(* IEC 61131-3 sources: ATCMcontrol_Engineering/src/COM/softing/fc/AddOns/Softing/4CPCTarget/Libs/ATCM_System, 28 files *)

(* ---- ClearLocalTaskErrno.st ---- *)
(*[[
    UserURL= "ATCM:ClearLocalTaskErrno.htm"
]]*)
(*
 *  ATCMControl Standard Function ClearLocalTaskErrno
 *  Purpose: Clears the error state of the given task.
 *)
FUNCTION ClearLocalTaskErrno
VAR_INPUT
    NAME : ANY_STRING;
END_VAR

overload (WSTRING) inline{((COM.softing.fc.CC.system.ITask)globals.getObject(%1.toLowerCase())).setErrorNumber(0)}

END_FUNCTION

(* ---- ClearTaskErrno.st ---- *)
(*[[
    UserURL= "ATCM:ClearTaskErrno.htm"
]]*)
(*
 *  ATCMControl Standard Function ClearTaskErrno
 *  Purpose: Clears the error state variable of the
 *           calling task. Error numbers <>0 signal an
 *           error.
 *)
FUNCTION ClearTaskErrno

inline{tc.setErrorNumber(0)}

END_FUNCTION

(* ---- ColdStartInstance.st ---- *)
(*
 * ATCMControl standard function ColdStartInstance
 * ----------------------------------------------------------------------------
 * PURPOSE: initialises all program, function block or structure instance members
 *          to their coldstart initial values. This includes also all nested
 *          function blocks and structs.
     *          The function returns if the initialisation is complete.
 *
 * EXAMPLE: StopLocalTask("Task1");
 *          ColdStartInstance("Prog1.myFB");
 *
 * NOTE:    It is recommended to stop the task(s) that operates on "Prog1.myFB"
 *          before calling ColdStartInstance.
 *
 * WARNING: use this function only rarely, it may take a long time to coldstart a
 *          huge and deeply nested instance, that could cause watchdog error in the
 *          calling task. Typically this function is used in a task that also
 *          starts/stops other Tasks and therefore SetSystemTask() was called to
 *          disable the watchdog anyway.
 *)
FUNCTION ColdStartInstance
VAR_INPUT
    instPath : WSTRING;
END_VAR

NATIVE
    int    i = 0;
    Object o = null;
    java.util.StringTokenizer st = new java.util.StringTokenizer(_instpath.toLowerCase(), ".");
    while (st.hasMoreTokens())
    {
        if (i == 0)
            o = ((ObjectDirectory)((FcObject)tc).getParent()).getObject(st.nextToken());
        else
            o = ((ObjectDirectory)o).getObject(st.nextToken());

        if (o == null)
            break;

        i++;
    }

    if (o == null || !(o instanceof ObjectDirectoryEx))
    {
        DebugManager.print("error E1056: ColdStartInstance: instance path '" + _instpath + "' does not exist.");
        return;
    }
    ObjectDirectoryEx od = (ObjectDirectoryEx)o;

    try{
        for(i=0; ;i++)
        {
            FcObject          fobj = od.getObjectByID(i);
            ObjectDescriptor  odescr = fobj.getOD();
            String            init = odescr.getInitString();

            if(init != null)
            {
                //DebugManager.print("vorher="+init);
                if(init.length()==0)
                {
                    init = null;//should not happen...
                }
                else if(init.charAt(0)=='%' && !(fobj instanceof COM.softing.fc.CC.system.StringVar))
                {
                    if(init.charAt(1)=='I')
                        continue;

                    int iPos = init.indexOf('|');
                    if(iPos>0 && iPos+1<init.length())
                    {
                        init = init.substring(iPos+1);
                    }
                    else
                    {
                        init = null;
                    }
                }
                //DebugManager.print("nachher="+init);
            }

            if (fobj instanceof FcBool)
            {
                ((FcBool)fobj).putBool(init==null ? false : init.equalsIgnoreCase("true"));
            }
            else if (fobj instanceof FcInt)
            {
                ((FcInt)fobj).putInt(init==null ? 0 : Integer.parseInt(init));
            }
            else if (fobj instanceof FcLong)
            {
              ((FcLong)fobj).putLong(init==null ? 0 : Long.parseLong(init));
            }
            else if (fobj instanceof FcDouble)
            {
              ((FcDouble)fobj).putDouble(init==null ? 0 : (new Double(init)).doubleValue());
            }
            else if (fobj instanceof FcString)
            {
              ((FcString)fobj).putString(init==null ? "" : init);
            }
            else if (fobj instanceof ObjectDirectoryEx)
            {
              _F_coldstartinstance(_instpath + "."+ fobj.getOD().getName(), globals, tc);
            }
            else
            {
               throw new ClassCastException("4CC : fatal error E0041: ColdStartInstance: unknown basic type class");
            }
        }
    }catch(ArrayIndexOutOfBoundsException e)
    {
        //normal end for loop: because there is no od.getLength() !!
    }
END_NATIVE;

END_FUNCTION

(* ---- DebugBreak.st ---- *)
(*[[
    UserURL= "ATCM:DebugBreak.htm"
]]*)
(*
 *  ATCMControl Standard Function DebugBreak
 *  Purpose: break into the debugger (only if one is attached)
 *)
FUNCTION DebugBreak
VAR_INPUT
    IN : BOOL; (* break only if IN = TRUE *)
END_VAR

inline{if(%1)tc.userBreak(this)}

END_FUNCTION

(* ---- EnableTaskStatistic.st ---- *)
(*[[
    UserURL= "ATCM:EnableTaskStatistic.htm"
]]*)
(*
 *  ATCMControl Standard Function EnableTaskStatistic
 *  Purpose: Enable/Disable the automatic task
 *  statistic output of all tasks.
 *  The default after a download or coldstart or
 *  warmstart is enable=true.
 *
 *  EnableTaskStatistic(true) : enable  task statistics
 *  EnableTaskStatistic(false): disable task statistics
 *)
FUNCTION EnableTaskStatistic
VAR_INPUT
    ENABLE     : BOOL;  (* enable/disable input *)
END_VAR

inline{tc.enableTaskStatistic(%1)}

END_FUNCTION

(* ---- GetComputerName.st ---- *)
(*
    Purpose: Gets the computername of the local PC.
*)
FUNCTION GetComputerName : WSTRING
NATIVE

    try{
        java.net.InetAddress  iaddr = java.net.InetAddress.getLocalHost();
        _getcomputername = iaddr.toString() ;//yields myPC1[.dhcp.softing.com]/129.26.193.3
        //if WinNT: strip .dhcp.softing.com (win2K does not need ??..)
        int idx = Math.min(_getcomputername.lastIndexOf('/'), _getcomputername.indexOf('.'));
        if(idx>0)
            _getcomputername = _getcomputername.substring(0, idx);
    }catch(java.net.UnknownHostException e)
    {
        _getcomputername = e.toString();
    }

END_NATIVE;

END_FUNCTION

(* ---- getCurrentDateAndTime.st ---- *)
(*[[
    UserURL= "ATCM:getCurrentDateAndTime.htm"
]]*)

FUNCTION getCurrentDateAndTime : DT

inline{java.lang.System.currentTimeMillis()}

END_FUNCTION

(* ---- GetLocalTaskErrno.st ---- *)
(*[[
    UserURL= "ATCM:GetLocalTaskErrno.htm"
]]*)
(*
 *  ATCMControl Standard Function GetLocalTaskErrno
 *  Purpose: get the task error number of the named task.
 *
 *  possible return values are (among others):
 *  NO_ERROR            = 0
 *  DEADLOCK_DETECTED   = 2
 *  RUNTIME_EXCEPTION   = 3
 *)
FUNCTION GetLocalTaskErrno : DINT
VAR_INPUT
    NAME : ANY_STRING;
END_VAR

overload DINT(WSTRING) inline{((COM.softing.fc.CC.system.ITask)globals.getObject(%1.toLowerCase())).itGetTaskErrNo()}

END_FUNCTION

(* ---- GetLocalTaskState.st ---- *)
(*[[
    UserURL= "ATCM:GetLocalTaskState.htm"
]]*)
(*
 *  ATCMControl Standard Function GetLocalTaskState
 *  Purpose: get the current task execution state of the named task.
 *
 *  possible return values are:
 *  STATE_ERROR       = -1
 *  STATE_ONCREATION  = 0
 *  STATE_STOPPED     = 1
 *  STATE_RUNNING     = 2
 *  STATE_BREAK       = 3
 *)
FUNCTION GetLocalTaskState : DINT
VAR_INPUT
    NAME : ANY_STRING;
END_VAR

overload DINT(WSTRING) inline{((COM.softing.fc.CC.system.ITask)globals.getObject(%1.toLowerCase())).itGetTaskState()}

END_FUNCTION

(* ---- GetTaskErrno.st ---- *)
(*[[
    UserURL= "ATCM:GetTaskErrno.htm"
]]*)
(*
 *  ATCMControl Standard Function GetTaskErrno
 *  Purpose: returns the last error number of the
 *           calling task. Error numbers <>0 signal an
 *           error.
 *)
FUNCTION GetTaskErrno : DINT

inline{tc.getErrorNumber()}

END_FUNCTION

(* ---- getTimeSinceSystemBoot.st ---- *)
(*[[
    UserURL= "ATCM:getTimeSinceSystemBoot.htm"
]]*)

FUNCTION getTimeSinceSystemBoot : TIME

inline{DebugManager.getSystemTime()}

END_FUNCTION

(* ---- OutputDebugString.st ---- *)
(*[[
    UserURL= "ATCM:OutputDebugString.htm"
]]*)
(*
 *  ATCMControl Standard Functionblock OutputDebugString
 *  Purpose: Write a string to the control's standard output
 *           and the log file. A new line character is added
 *           automatically.
 *)
FUNCTION OutputDebugString
VAR_INPUT
    STR        : ANY_STRING;     (* a one-line message to the user*)
END_VAR

overload (wstring) inline{DebugManager.print(%1 + "\n")}
(* TODO : string *)

END_FUNCTION

(* ---- ReadControlVarBOOL.st ---- *)
(*[[
]]*)
(*
 * ATCMControl standard function ReadControlVarBOOL
 * ----------------------------------------------------------------------------
 * PURPOSE: read from a named control variable.
 *
 * EXAMPLE: bValue := ReadControlVarBOOL("Prog1.myFB.aBool);
 *
 * RETURN:  if the function fails, a OutputDebugString
 *          is made and return is FALSE.
 *
 * WARNING: use this function only rarely, it is not efficient.
 *)
FUNCTION ReadControlVarBOOL : BOOL
VAR_INPUT
   sPath : WSTRING;     (* full qualified name of the variable to read *)
END_VAR

    ReadControlVarBOOL := FALSE;

    NATIVE
        int    i = 0;
        Object o = null;

        java.util.StringTokenizer st = new java.util.StringTokenizer(_spath.toLowerCase(), ".");
        while (st.hasMoreTokens())
        {
            if (i == 0)
                o = ((ObjectDirectory)((FcObject)tc).getParent()).getObject(st.nextToken());
            else
                o = ((ObjectDirectory)o).getObject(st.nextToken());

            if (o == null)
                break;

            i++;
        }

        if (o != null)
        {
            if (o instanceof FcBool)
            {
                _readcontrolvarbool = ((FcBool)o).getBool();
            }
            else
            {
                DebugManager.print("4C_Control(ReadControlVarBOOL): variable '" + _spath + "' is not a JAVA boolean.");
            }
        }
        else
        {
            DebugManager.print("4C_Control(ReadControlVarBOOL): variable '" + _spath + "' does not exist.");
        }
    END_NATIVE;
END_FUNCTION

(* $Header: /ABK4191 Liebherr Pruefstand-Modernisierung/4C-Basis/4C_Control/ReadControlVarBOOL.st 4     13.02.02 11:15 Go $
*----------------------------------------------------------------------------*
*
* =FILENAME            $Workfile: ReadControlVarBOOL.st $
*                       $Logfile: /ABK4191 Liebherr Pruefstand-Modernisierung/4C-Basis/4C_Control/ReadControlVarBOOL.st $
*
* =PROJECT             ABK4191 Liebherr Prüfstand-Modernisierung
*
* =COMPONENT           4C_Control Library
*
* =CURRENT      $Date: 13.02.02 11:15 $
*           $Revision: 4 $
*             $Author: Go $
*----------------------------------------------------------------------------*
*******************************************************************************
*)

(* ---- ReadControlVarDINT.st ---- *)
(*[[
]]*)
(*
 * ATCMControl standard function ReadControlVarDINT
 * ----------------------------------------------------------------------------
 * PURPOSE: read from a named control variable.
 *
 * EXAMPLE: aInt := ReadControlVarDINT("Prog1.myFB.aInt);
 *
 * RETURN:  if the function fails, a OutputDebugString
 *          is made and return is 0.
 *
 * WARNING: use this function only rarely, it is not efficient.
 *)
FUNCTION ReadControlVarDINT : DINT
VAR_INPUT
   sPath : WSTRING;     (* full qualified name of the variable to read *)
END_VAR

    ReadControlVarDINT := 0;

    NATIVE
        int    i = 0;
        Object o = null;

        java.util.StringTokenizer st = new java.util.StringTokenizer(_spath.toLowerCase(), ".");
        while (st.hasMoreTokens())
        {
            if (i == 0)
                o = ((ObjectDirectory)((FcObject)tc).getParent()).getObject(st.nextToken());
            else
                o = ((ObjectDirectory)o).getObject(st.nextToken());

            if (o == null)
                break;

            i++;
        }

        if (o != null)
        {
            if (o instanceof FcInt)
            {
                _readcontrolvardint = ((FcInt)o).getInt();
            }
            else
            {
                DebugManager.print("4C_Control(ReadControlVarDINT): variable '" + _spath + "' is not a JAVA int.");
            }
        }
        else
        {
            DebugManager.print("4C_Control(ReadControlVarDINT): variable '" + _spath + "' does not exist.");
        }
    END_NATIVE;
END_FUNCTION

(* ---- ReadControlVarLINT.st ---- *)
(*[[
]]*)
(*
 * ATCMControl standard function ReadControlVarLINT
 * ----------------------------------------------------------------------------
 * PURPOSE: read from a named control variable.
 *
 * EXAMPLE: aLreal := ReadControlVarLINT("Prog1.myFB.aLint");
 *
 * RETURN:  if the function fails, a corresponding
 *          OutputDebugString is made and return is 0.
 *
 * WARNING: use this function only rarely, it is not efficient.
 *)
FUNCTION ReadControlVarLINT : LINT
VAR_INPUT
   sPath : WSTRING;     (* full qualified name of the variable to read *)
END_VAR

    ReadControlVarLINT := 0;

    NATIVE
        int    i = 0;
        Object o = null;

        java.util.StringTokenizer st = new java.util.StringTokenizer(_spath.toLowerCase(), ".");
        while (st.hasMoreTokens())
        {
            if (i == 0)
                o = ((ObjectDirectory)((FcObject)tc).getParent()).getObject(st.nextToken());
            else
                o = ((ObjectDirectory)o).getObject(st.nextToken());

            if (o == null)
                break;

            i++;
        }

        if (o != null)
        {
            if (o instanceof FcLong)
            {
                _readcontrolvarlint = ((FcLong)o).getLong();
            }
            else
            {
                DebugManager.print("4C_Control(ReadControlVarLINT): variable '" + _spath + "' is not a JAVA long.");
            }
        }
        else
        {
            DebugManager.print("4C_Control(ReadControlVarLINT): variable '" + _spath + "' does not exist.");
        }
    END_NATIVE;

END_FUNCTION

(* ---- ReadControlVarLREAL.st ---- *)
(*[[
]]*)
(*
 * ATCMControl standard function ReadControlVarLREAL
 * ----------------------------------------------------------------------------
 * PURPOSE: read from a named control variable.
 *
 * EXAMPLE: aLreal := ReadControlVarLREAL("Prog1.myFB.aLreal");
 *
 * RETURN:  if the function fails, a OutputDebugString
 *          is made and return is 0.
 *
 * WARNING: use this function only rarely, it is not efficient.
 *)
FUNCTION ReadControlVarLREAL : LREAL
VAR_INPUT
   sPath : WSTRING;     (* full qualified name of the variable to read *)
END_VAR

    ReadControlVarLREAL := 0.0;

    NATIVE
        int    i = 0;
        Object o = null;

        java.util.StringTokenizer st = new java.util.StringTokenizer(_spath.toLowerCase(), ".");
        while (st.hasMoreTokens())
        {
            if (i == 0)
                o = ((ObjectDirectory)((FcObject)tc).getParent()).getObject(st.nextToken());
            else
                o = ((ObjectDirectory)o).getObject(st.nextToken());

            if (o == null)
                break;

            i++;
        }

        if (o != null)
        {
            if (o instanceof FcDouble)
            {
                _readcontrolvarlreal = ((FcDouble)o).getDouble();
            }
            else
            {
                DebugManager.print("4C_Control(ReadControlVarLREAL): variable '" + _spath + "' is not a JAVA double.");
            }
        }
        else
        {
            DebugManager.print("4C_Control(ReadControlVarLREAL): variable '" + _spath + "' does not exist.");
        }
    END_NATIVE;
END_FUNCTION

(* ---- ReadControlVarWSTRING.st ---- *)
(*[[
]]*)
(*
 * ATCMControl standard function ReadControlVarWSTRING
 * ----------------------------------------------------------------------------
 * PURPOSE: read from a named control variable.
 *
 * EXAMPLE: bStr := ReadControlVarWSTRING("Prog1.myFB.aStr");
 *
 * RETURN:  if the function fails, a OutputDebugString
 *          is made and return is "".
 *
 * WARNING: use this function only rarely, it is not efficient.
 *)
FUNCTION ReadControlVarWSTRING : WSTRING
VAR_INPUT
   sPath : WSTRING;     (* full qualified name of the variable to read *)
END_VAR

   ReadControlVarWSTRING  := "";

    NATIVE
        int    i = 0;
        Object o = null;
        java.util.StringTokenizer st = new java.util.StringTokenizer(_spath.toLowerCase(), ".");

        while (st.hasMoreTokens())
        {
            if (i == 0)
                o = ((ObjectDirectory)((FcObject)tc).getParent()).getObject(st.nextToken());
            else
                o = ((ObjectDirectory)o).getObject(st.nextToken());

            if (o == null)
                break;

            i++;
        }

        if (o != null)
        {
            if (o instanceof FcString)
            {
                _readcontrolvarwstring = ((FcString)o).getString();
            }
            else
            {
                DebugManager.print("4C_Control(ReadControlVarWSTRING): variable '" + _spath + "' is not a JAVA String.");
            }
        }
        else
        {
            DebugManager.print("4C_Control(ReadControlVarWSTRING): variable '" + _spath + "' does not exist.");
        }
    END_NATIVE;
END_FUNCTION

(* $Header: /ABK4191 Liebherr Pruefstand-Modernisierung/4C-Basis/4C_Control/ReadControlVarWSTRING.st 4     13.02.02 11:15 Go $
*----------------------------------------------------------------------------*
*
* =FILENAME            $Workfile: ReadControlVarWSTRING.st $
*                       $Logfile: /ABK4191 Liebherr Pruefstand-Modernisierung/4C-Basis/4C_Control/ReadControlVarWSTRING.st $
*
* =PROJECT             ABK4191 Liebherr Prüfstand-Modernisierung
*
* =COMPONENT           4C_Control Library
*
* =CURRENT      $Date: 13.02.02 11:15 $
*           $Revision: 4 $
*             $Author: Go $
*----------------------------------------------------------------------------*
*******************************************************************************
*)

(* ---- SetSystemTask.st ---- *)
(*[[
    UserURL= "ATCM:SetSystemTask.htm"
]]*)
(*
 *  ATCMControl Standard Function SetSystemTask
 *  Purpose: Declare this task to a system task.
 *           To be effective, this has to be the first
 *           statement of the program.
 *           System tasks are tasks that control
 *           other tasks via Start/StopLocalTask.
 *           A System Task will not be checked
 *           for dead-locks, so USE THIS CAREFULLY!
 *)
FUNCTION SetSystemTask

inline{tc.setSystemTask()}

END_FUNCTION

(* ---- SFCResetToInitialStep.st ---- *)
(*[[
    UserURL= "ATCM:SFCResetToInitialStep.htm"
]]*)
(*
 *  ATCMControl Standard Function SFCResetToInitialStep
 *  Purpose: reset SFC logic
 *)
FUNCTION SFCResetToInitialStep
VAR_INPUT
    ENABLE : BOOL; (* reset only if ENABLE = TRUE *)
END_VAR

inline{if(%1)this.resetToInitialStep()}

END_FUNCTION

(* ---- StartLocalTask.st ---- *)
(*[[
    UserURL= "ATCM:StartLocalTask.htm"
]]*)
(*
 *  ATCMControl Standard Function StartLocalTask
 *  Purpose: Put the named task to the running state.
 *)
FUNCTION StartLocalTask
VAR_INPUT
    NAME : ANY_STRING;
END_VAR

overload (WSTRING) inline{((COM.softing.fc.CC.system.ITask)globals.getObject(%1.toLowerCase())).itStartTask()}

END_FUNCTION

(* ---- StopLocalTask.st ---- *)
(*[[
    UserURL= "ATCM:StopLocalTask.htm"
]]*)
(*
 *  ATCMControl Standard Function StopLocalTask
 *  Purpose: Put the named task to the stopped state.
 *  WARNING: never try to stop the own task.
 *)
FUNCTION StopLocalTask
VAR_INPUT
    NAME : ANY_STRING;
END_VAR

overload (WSTRING) inline{((COM.softing.fc.CC.system.ITask)globals.getObject(%1.toLowerCase())).itStopTask()}

END_FUNCTION

(* ---- WriteControlVarBOOL.st ---- *)
(*[[
]]*)
(*
 * ATCMControl standard function WriteControlVarBOOL
 * ----------------------------------------------------------------------------
 * PURPOSE: write to a named control variable.
 *
 * EXAMPLE: bOk := WriteControlVarBOOL("Prog1.myFB.aBool, TRUE);
 *
 * RETURN:  if the function fails, a OutputDebugString
 *          is made and return is FALSE.
 *
 * WARNING: use this function only rarely, it is not efficient.
 *)
FUNCTION WriteControlVarBOOL : BOOL
VAR_INPUT
   sPath : WSTRING;       (* full qualified name of the variable to write *)
   bVal  : BOOL;          (* value to set *)
END_VAR

    WriteControlVarBOOL := FALSE;

    NATIVE
        int    i = 0;
        Object o = null;
        java.util.StringTokenizer st = new java.util.StringTokenizer(_spath.toLowerCase(), ".");

        while (st.hasMoreTokens())
        {
            if (i == 0)
                o = ((ObjectDirectory)((FcObject)tc).getParent()).getObject(st.nextToken());
            else
                o = ((ObjectDirectory)o).getObject(st.nextToken());

            if (o == null)
                break;

            i++;
        }

        if (o != null)
        {
            if (o instanceof FcBool)
            {
                ((FcBool)o).putBool(_bval);
                _writecontrolvarbool = true;
            }
            else
            {
                DebugManager.print("4C_Control(WriteControlVarBOOL): variable '" + _spath + "' is not a JAVA boolean.");
            }
        }
        else
        {
            DebugManager.print("4C_Control(WriteControlVarBOOL): variable '" + _spath + "' does not exist.");
        }
    END_NATIVE;
END_FUNCTION

(* $Header: /ABK4191 Liebherr Pruefstand-Modernisierung/4C-Basis/4C_Control/WriteControlVarBOOL.st 4     13.02.02 11:15 Go $
*----------------------------------------------------------------------------*
*
* =FILENAME            $Workfile: WriteControlVarBOOL.st $
*                       $Logfile: /ABK4191 Liebherr Pruefstand-Modernisierung/4C-Basis/4C_Control/WriteControlVarBOOL.st $
*
* =PROJECT             ABK4191 Liebherr Prüfstand-Modernisierung
*
* =COMPONENT           4C_Control Library
*
* =CURRENT      $Date: 13.02.02 11:15 $
*           $Revision: 4 $
*             $Author: Go $
*----------------------------------------------------------------------------*
*******************************************************************************
*)

(* ---- WriteControlVarDINT.st ---- *)
(*[[
]]*)
(*
 * ATCMControl standard function WriteControlVarDINT
 * ----------------------------------------------------------------------------
 * PURPOSE: write to a named control variable.
 *
 * EXAMPLE: bOk := WriteControlVarDINT("Prog1.myFB.aStr, "42");
 *
 * RETURN:  if the function fails, a OutputDebugString
 *          is made and return is FALSE.
 *
 * WARNING: use this function only rarely, it is not efficient.
 *)
FUNCTION WriteControlVarDINT : BOOL
VAR_INPUT
   sPath : WSTRING;       (* full qualified name of the variable to write *)
   iVal  : DINT;          (* value to set *)
END_VAR

    WriteControlVarDINT := FALSE;

    NATIVE
        int    i = 0;
        Object o = null;
        java.util.StringTokenizer st = new java.util.StringTokenizer(_spath.toLowerCase(), ".");

        while (st.hasMoreTokens())
        {
            if (i == 0)
                o = ((ObjectDirectory)((FcObject)tc).getParent()).getObject(st.nextToken());
            else
                o = ((ObjectDirectory)o).getObject(st.nextToken());

            if (o == null)
                break;

            i++;
        }

        if (o != null)
        {
            if (o instanceof FcInt)
            {
                ((FcInt)o).putInt(_ival);
                _writecontrolvardint = true;
            }
            else
            {
                DebugManager.print("4C_Control(WriteControlVarDINT): variable '" + _spath + "' is not a JAVA int.");
            }
        }
        else
        {
            DebugManager.print("4C_Control(WriteControlVarDINT): variable '" + _spath + "' does not exist.");
        }
    END_NATIVE;
END_FUNCTION

(* ---- WriteControlVarLINT.st ---- *)
(*[[
]]*)
(*
 * ATCMControl standard function WriteControlVarLINT
 * ----------------------------------------------------------------------------
 * PURPOSE: write to a named control variable.
 *
 * EXAMPLE: bOk := WriteControlVarLINT("Prog1.myFB.aLint", "42");
 *
 * RETURN:  if the function fails, a corresponding
 *          OutputDebugString is made and return is FALSE.
 *          If successfull the return value is TRUE.
 *
 * WARNING: use this function only rarely, it is not efficient.
 *)
FUNCTION WriteControlVarLINT : BOOL
VAR_INPUT
   sPath : WSTRING;       (* full qualified name of the variable to write *)
   iVal  : LINT;          (* value to set *)
END_VAR

    WriteControlVarLINT := FALSE;

    NATIVE
        int    i = 0;
        Object o = null;
        java.util.StringTokenizer st = new java.util.StringTokenizer(_spath.toLowerCase(), ".");

        while (st.hasMoreTokens())
        {
            if (i == 0)
                o = ((ObjectDirectory)((FcObject)tc).getParent()).getObject(st.nextToken());
            else
                o = ((ObjectDirectory)o).getObject(st.nextToken());

            if (o == null)
                break;

            i++;
        }

        if (o != null)
        {
            if (o instanceof FcLong)
            {
                ((FcLong)o).putLong(_ival);
                _writecontrolvarlint = true;
            }
            else
            {
                DebugManager.print("4C_Control(WriteControlVarLINT): variable '" + _spath + "' is not a JAVA int.");
            }
        }
        else
        {
            DebugManager.print("4C_Control(WriteControlVarLINT): variable '" + _spath + "' does not exist.");
        }
    END_NATIVE;

END_FUNCTION

(* ---- WriteControlVarLREAL.st ---- *)
(*[[
]]*)
(*
 * ATCMControl standard function WriteControlVarLREAL
 * ----------------------------------------------------------------------------
 * PURPOSE: write to a named control variable.
 *
 * EXAMPLE: bOk := WriteControlVarLREAL("Prog1.myFB.aStr, "42.0");
 *
 * RETURN:  if the function fails, a OutputDebugString
 *          is made and return is FALSE.
 *
 * WARNING: use this function only rarely, it is not efficient.
 *)
FUNCTION WriteControlVarLREAL : BOOL
VAR_INPUT
   sPath : WSTRING;       (* full qualified name of the variable to write *)
   lVal  : LREAL;         (* value to set *)
END_VAR

    WriteControlVarLREAL := FALSE;

    NATIVE
        int    i = 0;
        Object o = null;
        java.util.StringTokenizer st = new java.util.StringTokenizer(_spath.toLowerCase(), ".");

        while (st.hasMoreTokens())
        {
            if (i == 0)
                o = ((ObjectDirectory)((FcObject)tc).getParent()).getObject(st.nextToken());
            else
                o = ((ObjectDirectory)o).getObject(st.nextToken());

            if (o == null)
                break;

            i++;
        }

        if (o != null)
        {
            if (o instanceof FcDouble)
            {
                ((FcDouble)o).putDouble(_lval);
                _writecontrolvarlreal = true;
            }
            else
            {
                DebugManager.print("4C_Control(WriteControlVarLREAL): variable '" + _spath + "' is not a JAVA double.");
            }
        }
        else
        {
            DebugManager.print("4C_Control(WriteControlVarLREAL): variable '" + _spath + "' does not exist.");
        }
    END_NATIVE;
END_FUNCTION

(* ---- WriteControlVarWSTRING.st ---- *)
(*[[
]]*)
(*
 * ATCMControl standard function WriteControlVarWSTRING
 * ----------------------------------------------------------------------------
 * PURPOSE: write to a named control variable.
 *
 * EXAMPLE: bOk := WriteControlVarWSTRING("Prog1.myFB.aStr, "42");
 *
 * RETURN:  if the function fails, a OutputDebugString
 *          is made and return is FALSE.
 *
 * WARNING: use this function only rarely, it is not efficient.
 *)
FUNCTION WriteControlVarWSTRING : BOOL
VAR_INPUT
   sPath : WSTRING;       (* full qualified name of the variable to write *)
   sVal  : WSTRING;       (* value to set *)
END_VAR

    WriteControlVarWSTRING  := FALSE;

    NATIVE
        int    i = 0;
        Object o = null;
        java.util.StringTokenizer st = new java.util.StringTokenizer(_spath.toLowerCase(), ".");

        while (st.hasMoreTokens())
        {
            if (i == 0)
                o = ((ObjectDirectory)((FcObject)tc).getParent()).getObject(st.nextToken());
            else
                o = ((ObjectDirectory)o).getObject(st.nextToken());

            if (o == null)
                break;

            i++;
        }

        if (o != null)
        {
            if (o instanceof FcString)
            {
                ((FcString)o).putString(_sval);
                _writecontrolvarwstring = true;
            }
            else
            {
                DebugManager.print("4C_Control(WriteControlVarWSTRING): variable '" + _spath + "' is not a JAVA String.");
            }
        }
        else
        {
            DebugManager.print("4C_Control(WriteControlVarWSTRING): variable '" + _spath + "' does not exist.");
        }
    END_NATIVE;
END_FUNCTION

(* ---- fc_debug.st ---- *)
(*[[
    UserURL= "ATCM:FC_DEBUG.htm"
]]*)

(*
 *  ATCMControl Standard Functionblock FC_DEBUG
 *  Purpose: Debug Output
 *)
FUNCTION_BLOCK FC_DEBUG
VAR_INPUT
    ENABLE     : BOOL:=TRUE;  (* enable output with this inst  *)
    STR        : WSTRING;     (* a one-line message to the user*)
END_VAR

IF ENABLE THEN
    NATIVE
        DebugManager.print(_str.getString() + '\n');
    END_NATIVE;
END_IF;

END_FUNCTION_BLOCK

(* ---- SignalError.st ---- *)
(*[[
    UserURL= "ATCM:SignalError.htm"
]]*)
(*
 *  ATCMControl Standard Functionblock SignalError
 *  Purpose: Send Task to Error State
 *
 *  if enable=TRUE and errno<>0 then
 *    the current task is stopped.
 *)
FUNCTION_BLOCK SignalError

VAR_INPUT
    ENABLE     : BOOL:=TRUE;  (* enable this inst *)
    ERRNO      : DINT:=0;     (* error number *)
END_VAR

IF ENABLE AND ERRNO<>0 THEN
    NATIVE
        DebugManager.print("4CC : error E1000: SignalError(ERRNO=" + _errno.getInt() +")\n");
        Thread.dumpStack();
        tc.errorTask(_errno.getInt());
    END_NATIVE;
END_IF;

END_FUNCTION_BLOCK
